{attribute addProperty BoxType "AX5206-0000-0200-0200"}
{attribute addProperty Id "AT_xAT %I*ARRAY[0..1] OF AT_15FCA3A6160200MDTAT %Q*ARRAY[0..1] OF MDT_C2B17B7F96120WcStateAT %I*WcState_98A4DF7520.250InfoDataAT %I*InfoData_81099714160200"}
{attribute addProperty CRC "3871957761"}
{attribute addProperty SizeInBites "418"}
{attribute addProperty SizeInBytes "52.25"}
TYPE AX5206_7BA23180 :
STRUCT
	{attribute addProperty Name "AT"}
	AT_x : ARRAY[0..1] OF AT_15FCA3A6;
	{attribute addProperty Name "MDT"}
	MDT : ARRAY[0..1] OF MDT_C2B17B7F;
	{attribute addProperty Name "WcState"}
	WcState : WcState_98A4DF75;
	{attribute addProperty Name "InfoData"}
	InfoData : InfoData_81099714;
END_STRUCT
END_TYPE

(* stored: Version 1.2.0.0, ProductVersion 3.1.4024.9
   DUT AX5206_7BA23180: Id {299d26ee-edd5-4e5a-8d76-27aea1ad2cfc} *)
